INTERFACE I_OPCUA_Disconnect

METHOD start : BOOL
VAR_INPUT
    Execute           : BOOL;
    ConnectionHdl     : DWORD;     
    Timeout           : TIME := DEFAULT_ADS_TIMEOUT; 
END_VAR 
VAR_OUTPUT
    Done        : BOOL;
    Busy        : BOOL;
    Error       : BOOL;
    ErrorID     : DWORD;
END_VAR
END_METHOD

END_INTERFACE

(* stored: Version 1.1.0.1, ProductVersion 3.1.4024.9
   Itf I_OPCUA_Disconnect: Id {64f61633-4c3c-4f0f-8db9-d6021f05b6db}
   Method start: Id {08488aa1-4d81-4a4d-86b9-5bacc9a0a85a} *)
